FUNCTION_BLOCK StateProxy IMPLEMENTS I_Debug
VAR_INPUT
END_VAR
VAR_OUTPUT
END_VAR
VAR
END_VAR

//FB_Init is always available implicitly and it is used primarily for initialization.
//The return value is not evaluated. For a specific influence, you can also declare the
//methods explicitly and provide additional code there with the standard initialization
//code. You can evaluate the return value.
METHOD FB_Init: BOOL
VAR_INPUT
    bInitRetains: BOOL; // TRUE: the retain variables are initialized (reset warm / reset cold)
    bInCopyCode: BOOL;  // TRUE: the instance will be copied to the copy code afterward (online change)   

	iState		: I_State;
	refState	: REFERENCE TO I_State;
END_VAR
IF NOT __ISVALIDREF(refState) THEN
	DebugMsg(THIS^, 'Ref = 0!');
	RETURN;
END_IF

IF iState = 0 THEN
	DebugMsg(THIS^, 'Itf = 0!');
	RETURN;
END_IF

IF refState <> 0 THEN
	DebugMsg(THIS^, 'Ref itf should be unassigned!');
	RETURN;
END_IF

refState := iState;
END_METHOD

END_FUNCTION_BLOCK

(* stored: Version 1.1.0.1
   POU StateProxy: Id {3adaacfd-2bb2-42d1-b426-c26bd852962c}, SpecialFunc None
   Method FB_init: Id {f592e959-64f6-4f51-99ce-3f86d7875f50} *)
